FUNCTION_BLOCK T_RoboConnect_MoveJWrongCount_ReturnsFalse EXTENDS T_UnitTestBase
VAR
  robot : T_MockRoboConnect;
  targets : ARRAY [1..4] OF LREAL;
  expected : BOOL := FALSE;
  actual : BOOL := TRUE;
END_VAR

actual := robot.MoveJ(targets);
assertion.AssertEquals_BOOL(expected, actual, 'actual := robot.MoveJ(targets)');
TestFinished();

END_FUNCTION_BLOCK

(* stored: Version 1.1.0.1
   POU T_TcRobot_MoveJWrongCount_ReturnsFalse: Id {663f15a1-4e03-43a0-bf7f-425e2d583689}, SpecialFunc None *)
